{region '#Template'}
	{attribute 'Version' := '1.2.2.0'}
	{attribute 'Tags' := '"LCID": "1031", "Text": "AC, Setpoint, Temperatur, Cascade control"'}
	{attribute 'Tags' := '"LCID": "1033", "Text": "AC, Setpoint, Temperatur, Cascade control"'}
	{attribute 'Using' := '"Type": "Template", "URI": "BA2_Param"'}
	{attribute 'Using' := '"Type": "Template", "URI": "E_BA_MdltCmd"'}
	{attribute 'Using' := '"Type": "Template", "URI": "E_BA_AC_SelSpErc"'}
	{attribute 'Description' := '"LCID": "1031", "Text": "Temperatur Kaskadenregelung"'}
	{attribute 'Description' := '"LCID": "1033", "Text": "Temperature Cascade control"'}
{endregion}
FUNCTION_BLOCK FB_BA_AC_TCasCtrl_01 EXTENDS FB_BA_AggregateM
VAR_INPUT
	fSpTRm					: REAL;
	fTRm					: REAL;
END_VAR                                                         	
VAR_OUTPUT                                                      	
	fSpHtg					: REAL;
	fSpCol					: REAL;
	fSpErc					: REAL;
	fMax					: REAL;
	fMin					: REAL;
	bOn						: BOOL;	
END_VAR
VAR
	eOpMode					: REFERENCE TO E_BA_MdltCmd		REF= nActiveVal;
END_VAR
VAR_INPUT CONSTANT
	SpHtg					: FB_BA_AV_Op;									
	SpCol					: FB_BA_AV_Op;																				  
	SpErc					: FB_BA_AV_Op;		
	Ctrl					: FB_BA_Loop;	
END_VAR
VAR
	MuxEnSeqCtrl			: FB_BA_MMUX_B04;
	MuxSpHtg				: FB_BA_MMUX_R04;
	MuxSpCol				: FB_BA_MMUX_R04;
	MuxSpErc				: FB_BA_MMUX_R04;
END_VAR
VAR // added by the converter: edge detectors and wires of the graphical bodies
    _w1 : BOOL;
    _w2 : REAL;
END_VAR

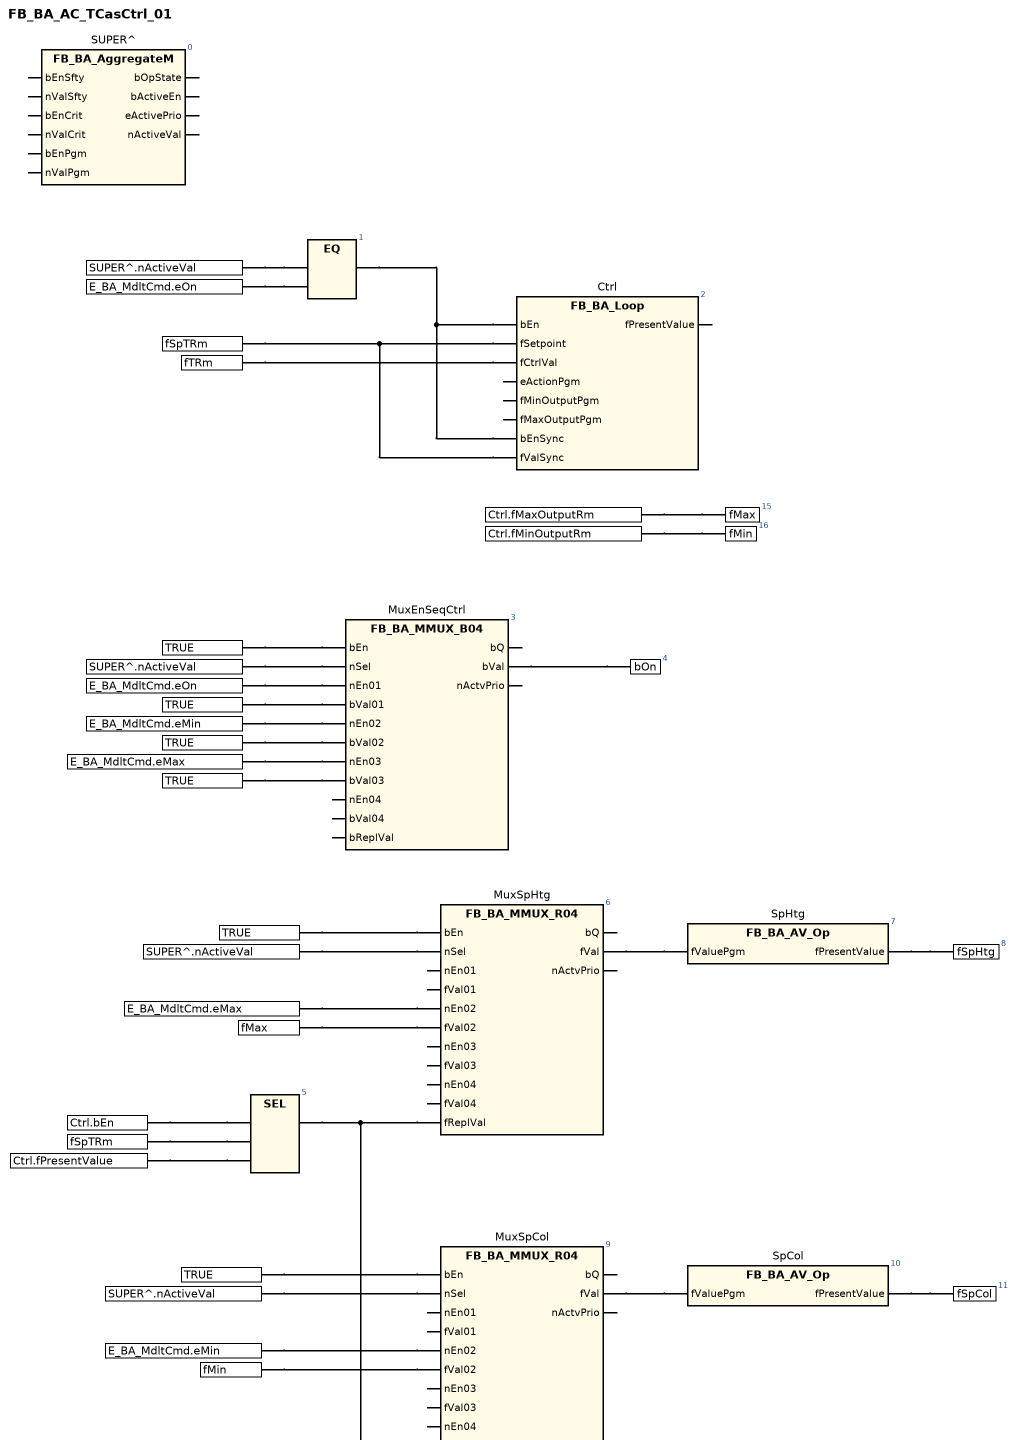
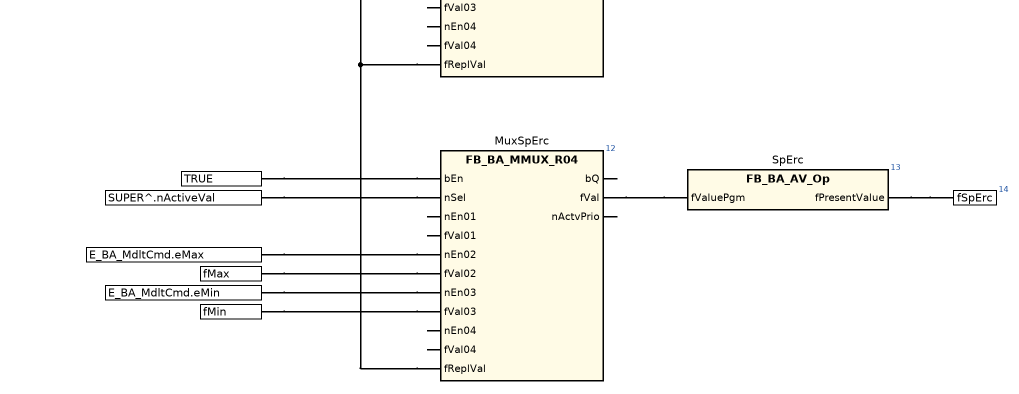
SUPER^(); // FB_BA_AggregateM
_w1 := SUPER^.nActiveVal = E_BA_MdltCmd.eOn;
Ctrl(bEn := _w1, fSetpoint := fSpTRm, fCtrlVal := fTRm, bEnSync := _w1, fValSync := fSpTRm); // FB_BA_Loop
MuxEnSeqCtrl(
    bEn := TRUE,
    nSel := SUPER^.nActiveVal,
    nEn01 := E_BA_MdltCmd.eOn,
    bVal01 := TRUE,
    nEn02 := E_BA_MdltCmd.eMin,
    bVal02 := TRUE,
    nEn03 := E_BA_MdltCmd.eMax,
    bVal03 := TRUE); // FB_BA_MMUX_B04
bOn := MuxEnSeqCtrl.bVal;
_w2 := SEL(Ctrl.bEn, fSpTRm, Ctrl.fPresentValue);
MuxSpHtg(bEn := TRUE, nSel := SUPER^.nActiveVal, nEn02 := E_BA_MdltCmd.eMax, fVal02 := fMax, fReplVal := _w2); // FB_BA_MMUX_R04
SpHtg(fValuePgm := MuxSpHtg.fVal); // FB_BA_AV_Op
fSpHtg := SpHtg.fPresentValue;
MuxSpCol(bEn := TRUE, nSel := SUPER^.nActiveVal, nEn02 := E_BA_MdltCmd.eMin, fVal02 := fMin, fReplVal := _w2); // FB_BA_MMUX_R04
SpCol(fValuePgm := MuxSpCol.fVal); // FB_BA_AV_Op
fSpCol := SpCol.fPresentValue;
MuxSpErc(
    bEn := TRUE,
    nSel := SUPER^.nActiveVal,
    nEn02 := E_BA_MdltCmd.eMax,
    fVal02 := fMax,
    nEn03 := E_BA_MdltCmd.eMin,
    fVal03 := fMin,
    fReplVal := _w2); // FB_BA_MMUX_R04
SpErc(fValuePgm := MuxSpErc.fVal); // FB_BA_AV_Op
fSpErc := SpErc.fPresentValue;
fMax := Ctrl.fMaxOutputRm;
fMin := Ctrl.fMinOutputRm;

METHOD FB_init : BOOL
VAR_INPUT
	bInitRetains : BOOL; // if TRUE, the retain variables are initialized (warm start / cold start)
	bInCopyCode : BOOL;  // if TRUE, the instance afterwards gets moved into the copy code (online change)
END_VAR
SpHtg.iParent						:= THIS^;
SpHtg.iLabel						:= LblCmpAC.TCasCtrl_SpHtg;			
SpHtg.sObjectName					:= '{Idx=01}';								 	 
SpHtg.eUnit							:= E_BA_Unit.eTemperature_DegreesCelsius;  
SpHtg.fCOVIncrement					:= BA2_Param.fDefCOVIncrement;							

SpCol.iParent						:= THIS^;
SpCol.iLabel						:= LblCmpAC.TCasCtrl_SpCol;			
SpCol.sObjectName					:= '{Idx=02}';								 	 
SpCol.eUnit							:= E_BA_Unit.eTemperature_DegreesCelsius;  
SpCol.fCOVIncrement					:= BA2_Param.fDefCOVIncrement;							
									
SpErc.iParent						:= THIS^;
SpErc.iLabel						:= LblCmpAC.TCasCtrl_SpErc;			
SpErc.sObjectName					:= '{Idx=03}';								 	 
SpErc.eUnit							:= E_BA_Unit.eTemperature_DegreesCelsius;  
SpErc.fCOVIncrement					:= BA2_Param.fDefCOVIncrement;							

Ctrl.iParent						:= THIS^;
Ctrl.iLabel							:= LblCmpAC.TCasCtrl_Ctrl; 
Ctrl.sObjectName					:= '{Idx=01}';
Ctrl.eOpMode						:= BA2_Param.nLoop_DefOpMode;								 	 										 
Ctrl.eOutputUnit					:= E_BA_Unit.eTemperature_DegreesCelsius;
Ctrl.eActionRm						:= E_BA_Action.eReverse;
Ctrl.fProportionalConstant			:= 1.5;
Ctrl.fIntegralConstant				:= 360;
Ctrl.fDerivativeConstant			:= 0;
Ctrl.fMaxOutputRm 					:= 32;
Ctrl.fMinOutputRm					:= 16;
Ctrl.fCOVIncrement					:= 0;
Ctrl.nDampConstant					:= 0;
Ctrl.fNeutralZone					:= 0;
END_METHOD

END_FUNCTION_BLOCK

(* stored: Version 1.1.0.1, ProductVersion 3.1.4024.9
   POU FB_BA_AC_TCasCtrl_01: Id {bc1a9304-2d21-4853-bfb6-7def207edbc7}, SpecialFunc None
   Method FB_init: Id {384a0b3e-897d-4d36-96e9-6ad8e9b68cda} *)
